PROGRAM PRG_Test
VAR
END_VAR


	TcUnit.RUN_IN_SEQUENCE ();

END_PROGRAM

(* stored: Version 1.1.0.1
   POU PRG_Test: Id {1d1ad101-c2d4-0277-1bb3-7445680eebd7}, SpecialFunc None *)
